FUNCTION_BLOCK Room_Ctx IMPLEMENTS I_Room
VAR_STAT
	_nNextRoom	: UDINT;
END_VAR
VAR_INPUT
	io			: Room_Ctx_Io;
	hmi			: Room_Ctx_Hmi;
	priv		: Room_Ctx_Priv;
END_VAR
VAR_OUTPUT
	state		: Room_Ctx_States;	
END_VAR

//FB_Init is always available implicitly and it is used primarily for initialization.
//The return value is not evaluated. For a specific influence, you can also declare the
//methods explicitly and provide additional code there with the standard initialization
//code. You can evaluate the return value.
METHOD FB_Init: BOOL
VAR_INPUT
    bInitRetains: BOOL; // TRUE: the retain variables are initialized (reset warm / reset cold)
    bInCopyCode: BOOL;  // TRUE: the instance will be copied to the copy code afterward (online change)
END_VAR
_nNextRoom := _nNextRoom + 1;
hmi.nId := _nNextRoom;
END_METHOD

METHOD GoFault
VAR_INPUT
	sErrorText		: Str;
END_VAR
hmi.sErrorText := sErrorText;
state.iMgr.Request(state.iFault);
END_METHOD

METHOD GoHeat
IF NOT priv.bActive THEN
	RETURN;
END_IF

io.bOpenValves := TRUE;
END_METHOD

METHOD GoIdle
IF NOT priv.bActive THEN
	RETURN;
END_IF

state.iMgr.Request(state.iIdle);
END_METHOD

PROPERTY Id : UDINT
GET
Id := hmi.nId;
END_GET
END_PROPERTY

PROPERTY IsActive : BOOL
GET
IsActive := priv.bActive;
END_GET
END_PROPERTY

PROPERTY IsClosed : BOOL
GET
IsClosed := io.bValvesClosed;
END_GET
END_PROPERTY

PROPERTY IsOpen : BOOL
GET
IsOpen := io.bValvesOpen;
END_GET
END_PROPERTY

PROPERTY IsReady : BOOL
GET
IsReady := priv.bReady;
END_GET
END_PROPERTY

PROPERTY Timeout : TIME
GET
Timeout := UDINT_TO_TIME(hmi.nTimeout * 1000 * 60);
END_GET
END_PROPERTY

END_FUNCTION_BLOCK

(* stored: Version 1.1.0.1
   POU Room_Ctx: Id {6599786c-ba93-4fed-b30a-839e05cc02d4}, SpecialFunc None
   Folder _: Id {93023407-6fce-4cd4-a59f-f4e5ea04c3a7}
   Folder Flags: Id {9bd30358-ab44-46bf-81aa-ba6b3185935e}
   Folder Request: Id {58538f0c-0c0f-4a71-8112-ce2d7fd2ab3d}
   Method FB_init: Id {ca22bbab-be21-4373-9409-1f9b1007feee}
   Method GoFault: Id {58bcbc1a-fac3-413a-a2a2-69cf90b35fc2}
   Method GoHeat: Id {2ef519f7-2d21-4fe3-a50b-7c53dc7ef0e6}
   Method GoIdle: Id {a7b9d657-00fa-45e9-baeb-af69e6018523}
   Property Id: Id {cab61793-e91a-43d3-b4f1-43fa7063eb1d}
   Get Get: Id {0db4bec7-83f4-40cb-a9f0-f42887b91727}
   Property IsActive: Id {05099b11-7bf8-4c59-9cb6-a7bb7b3a2db4}
   Get Get: Id {9fda7680-eecb-4790-855c-e58914c1503a}
   Property IsClosed: Id {8201ff4f-9b53-446e-b50e-9f3ccbca46fc}
   Get Get: Id {860a5c51-d17a-487c-8cbf-c0e50bf3bb19}
   Property IsOpen: Id {363ee4e3-517b-4e8e-a8ef-3e40d440e3f6}
   Get Get: Id {19a270b5-a546-429e-9caa-5fce82d24831}
   Property IsReady: Id {faede1ff-4852-4edb-be53-dba65663064d}
   Get Get: Id {9ff15937-25cb-474e-b7f4-31a6db2c8096}
   Property Timeout: Id {eecc649b-322a-4026-a5ac-c0aea4a056f0}
   Get Get: Id {2bf87570-2da5-4e3e-8bee-0d0856799639} *)
